// TIA Portal V18 export
FUNCTION_BLOCK "_DOOORS_fb"   // FB72, FBD
{ S7_Optimized_Access := 'TRUE' }
VERSION : 0.1
// stored: AutoNumber true, IsIECCheckEnabled false, IsRetainMemResEnabled false, MemoryReserve 100, SetENOAutomatically false, UDAEnableTagReadback false
   VAR_INPUT
      xBtnOpen : Bool;
      xBtnClose : Bool;
      allowedNotAuto : Bool;
      allowedCloseLightBrrier : Bool;
      allowedCloseManipulator : Bool;
      xClosed : Bool;
      xOpen : Bool;
   END_VAR
   VAR_OUTPUT
      yCmdOpen : Bool;
      yCmdClose : Bool;
      sOpen : Bool;
      sClosed : Bool;
      wn_Auto : Bool;
      wnLightbarrier : Bool;
      wnManipulatorClose : Bool;
   END_VAR
   VAR_IN_OUT
      yBeepCosedResetMe : Bool;
   END_VAR
   VAR
      memOpen : Bool;
      memClosed : Bool;
      memopn : Bool;
      memopn1 : Bool;
      memClosed1 : Bool;
   END_VAR
   VAR_TEMP   // added for the SCL form of the ladder/FBD networks
      _w1 : Bool;
      _w2 : Bool;
   END_VAR
BEGIN

REGION Network 1
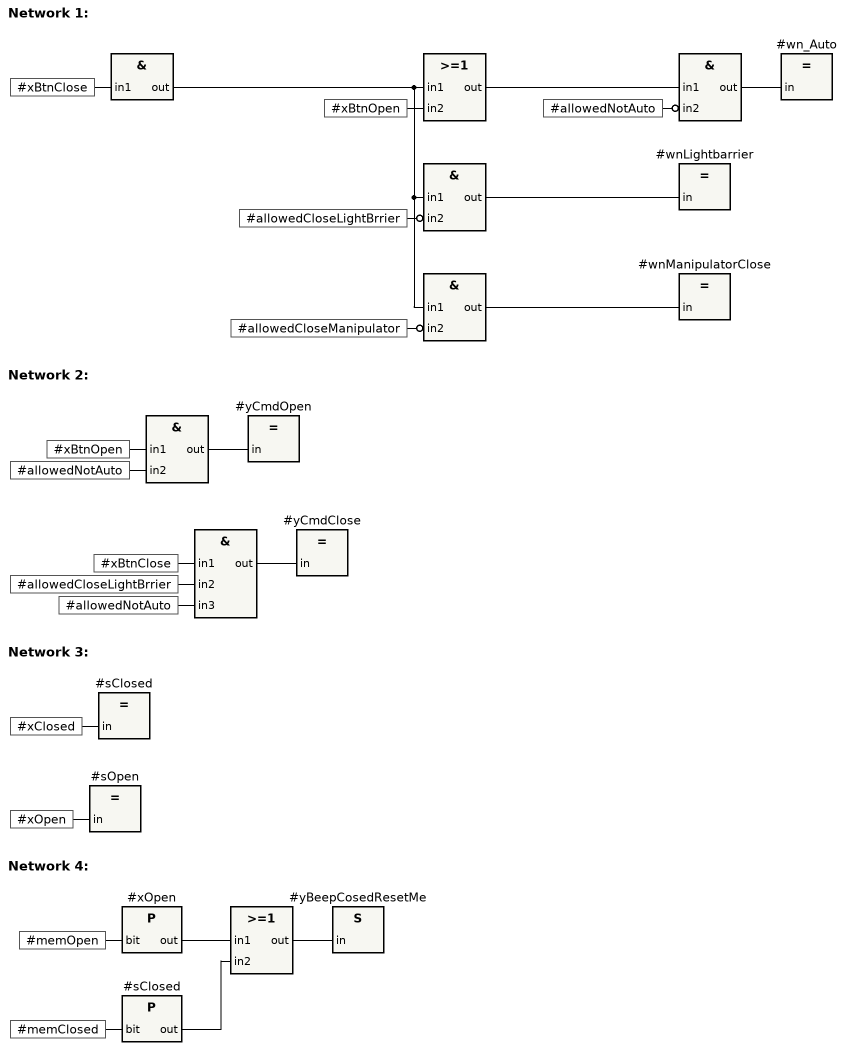
   #wn_Auto := (#xBtnClose OR #xBtnOpen) AND NOT #allowedNotAuto;
   #wnLightbarrier := #xBtnClose AND NOT #allowedCloseLightBrrier;
   #wnManipulatorClose := #xBtnClose AND NOT #allowedCloseManipulator;
END_REGION

REGION Network 2
   #yCmdOpen := #xBtnOpen AND #allowedNotAuto;
   #yCmdClose := #xBtnClose AND #allowedCloseLightBrrier AND #allowedNotAuto;
END_REGION

REGION Network 3
   #sClosed := #xClosed;
   #sOpen := #xOpen;
END_REGION

REGION Network 4
   #_w1 := #xOpen AND NOT #memOpen;   // rising edge of #xOpen
   #memOpen := #xOpen;
   #_w2 := #sClosed AND NOT #memClosed;   // rising edge of #sClosed
   #memClosed := #sClosed;
   IF #_w1 OR #_w2 THEN #yBeepCosedResetMe := TRUE; END_IF;
END_REGION
END_FUNCTION_BLOCK
